TYPE TRunCmdPearling :
	(
		RCP_None,
		RCP_Pearl,
		RCP_ChangeChuck,
		RCP_CheckSharpen
	);
END_TYPE

(* stored: Version 1.1.0.1, ProductVersion 3.1.4022.12
   DUT TRunCmdPearling: Id {7ad051bb-179c-49dc-9707-6b555341197b} *)
